PROGRAM PRG_PMPS
VAR
    fbArbiterIO: FB_SubSysToArbiter_IO;

    {attribute 'TcLinkTo' := 'TIIB[PMPS_PRE]^IO Outputs^FFO'}
    FFO AT %Q*:BOOL; //temp code until faults are in MPS crate
END_VAR

GVL.fbFastFaultOutput1.Execute(i_xVeto := (PMPS_GVL.stCurrentBeamParameters.aVetoDevices[PMPS.K_Stopper.MR1K1_IN]
                                      AND NOT PMPS_GVL.stCurrentBeamParameters.aVetoDevices[PMPS.K_Stopper.MR1K1_OUT])
                                       OR PMPS_GVL.stCurrentBeamParameters.aVetoDevices[PMPS.K_Stopper.MR1K3_OUT]
                                      AND NOT PMPS_GVL.stCurrentBeamParameters.aVetoDevices[PMPS.K_Stopper.MR1K1_IN]);
fbArbiterIO(
    i_bVeto := (PMPS_GVL.stCurrentBeamParameters.aVetoDevices[PMPS.K_Stopper.MR1K1_IN]
                                      AND NOT PMPS_GVL.stCurrentBeamParameters.aVetoDevices[PMPS.K_Stopper.MR1K1_OUT])
                                       OR PMPS_GVL.stCurrentBeamParameters.aVetoDevices[PMPS.K_Stopper.MR1K3_OUT]
                                      AND NOT PMPS_GVL.stCurrentBeamParameters.aVetoDevices[PMPS.K_Stopper.MR1K1_IN],
    Arbiter:=GVL.fbArbiter1,
    fbFFHWO:=GVL.fbFastFaultOutput1);

GVL.fbArbiter1.AddRequest(nReqID := 16#FAF7, stReqBp := PMPS_GVL.cstFullBeam, sDevName := 'plc-kfe-txi-mot');

//TEMP FFO to arbiter
FFO:= GVL.fbFastFaultOutput1.q_xFastFaultOut;

END_PROGRAM

(* stored: Version 1.1.0.1, ProductVersion 3.1.4024.6
   POU PRG_PMPS: Id {dff18baf-d3c9-4cb4-be04-4a60c54f1a90}, SpecialFunc None *)
